(* IEC 61131-3 sources: SRCI/RobotLibrary/Library/POUs/Additional/MC_UnitMeasurement, 1 file *)

(* ---- MC_UnitMeasurementFB.st ---- *)
/// Measure the length of objects in the cartesian space, execution time for specified section of a job or signal output time of a specified signal
FUNCTION_BLOCK MC_UnitMeasurementFB EXTENDS RobotLibraryBaseEnableFB
// -------------------------------------------------------------------------
//  SRCI Robot Library
// -------------------------------------------------------------------------
//
//  Object:      UnitMeasurementFB
//  Author:      Thorsten Brach
//  Date:        2024-06-01
//
//  Description:
//
//
//  Copyright:
//    (C) 2024 Thorsten Brach. All rights reserved
//             Licensed under the LGPL-3.0 license.
//
//  Disclaimer:
//    This project is provided without any guarantee and can be used for
//    private and commercial purposes. Any use is at the user’s
//    own risk and responsibility.
//
// -------------------------------------------------------------------------
VAR_INPUT
  /// command results
  ParCmd            : UnitMeasurementParCmd;
END_VAR

VAR_OUTPUT
  /// Command is transferred and confirmed by the RC
  CommandBuffered   : BOOL;
  /// Receiving of input parameter values has been acknowledged by RC
  ParameterAccepted : BOOL;
  /// command results
  OutCmd            : UnitMeasurementOutCmd;
END_VAR

VAR
  /// internal copy of command parameter
 _parCmd            : UnitMeasurementParCmd;
  /// command data to send
 _command           : UnitMeasurementSendData;
  /// response data received
 _response          : UnitMeasurementRecvData;
  /// measurement number
 _measurementNo     : USINT;
END_VAR

  SUPER^(AxesGroup := AxesGroup);

END_FUNCTION_BLOCK

METHOD INTERNAL CheckAddParameter : BOOL
VAR_INPUT
  /// Payload pointer
  PayloadPtr : UDINT;
END_VAR
VAR
  /// Payload as byte array
  Payload    : ARRAY [1..SIZEOF(_command)] OF BYTE;
  /// Null Byte array
  Null       : ARRAY [1..SIZEOF(_command)] OF BYTE;
  /// Data length to compare
  DataLen    : UDINT;
END_VAR

  // Payload pointer must be decreased by one byte, because ADR(Payload) is already one byte !
  PayloadPtr := LIMIT (0, PayloadPtr - 1, SIZEOF(Payload) -1);
  // Convert command struct to payload array
  SysDepMemCpy( pDest := ADR(Payload), pSrc := ADR(_command), DataLen := SIZEOF(_command));
  // Calculate the data length to compare - at least one byte must be compared !
  DataLen := LIMIT(1, SIZEOF(Payload) - PayloadPtr, SIZEOF(Payload));
  // Compare Payload-Array with Null-Byte-Array
  CheckAddParameter := SysDepMemCmp( pData1 := ADR(Payload) + PayloadPtr , pData2 := ADR(Null), DataLen := DataLen) <>  RobotLibraryConstants.OK ;

END_METHOD

METHOD PROTECTED CheckFunctionSupported : BOOL
VAR_IN_OUT
  /// Robot assignment of function
  AxesGroup : AxesGroup;
END_VAR

  CheckFunctionSupported := AxesGroup.State.RobotData.RCSupportedFunctions.UnitMeasurement;

  IF ( NOT CheckFunctionSupported )
  THEN
    // call base implementation for set error and create log entry
    SUPER^.CheckFunctionSupported(AxesGroup := AxesGroup);
  END_IF

END_METHOD

METHOD PROTECTED CheckParameterChanged : BOOL
VAR_IN_OUT
  /// Robot assignment of function
  AxesGroup    : AxesGroup;
END_VAR

  // Check ParCmd Size is > 0, because MemCmp does not work correctly with size = 0
  IF (SIZEOF(ParCmd) = 0) OR (_stepCmd = 0)
  THEN
    RETURN;
  END_IF

  // compare memory
  _parameterChanged := ( SysDepMemCmp(pData1 := ADR(ParCmd), pData2 := ADR(_parCmd), DataLen := SIZEOF(ParCmd)) <> RobotLibraryConstants.OK );

  // check parameter valid ?
  _parameterValid   := CheckParameterValid( AxesGroup := AxesGroup );

  IF ((  _parameterChanged        )  AND
      (  _parameterValid          )) OR
      (  _parameterUpdateInternal )
  THEN
    // reset internal flag for send parameter update
   _parameterUpdateInternal := FALSE;
    // update internal copy of parameters
   _parCmd := ParCmd;
    // inc parameter sequence
   _command.ParSeq := _command.ParSeq + 1;
    // update command data
    CommandData := CreateCommandPayload(AxesGroup := AxesGroup); // ( Access via reference to rCommandFB in ACR )
    // notify active command register
    AxesGroup.Acyclic.ActiveCommandRegister.NotifyParameterChanged := _uniqueID;
    // Reset parameter accepted flag
    ParameterAccepted := FALSE;
  END_IF

END_METHOD

METHOD PROTECTED CheckParameterValid : BOOL
VAR_IN_OUT
  /// Robot assignment of function
  AxesGroup : AxesGroup;
END_VAR

  CheckParameterValid := TRUE;

  // Check ParCmd.TriggerMode valid ?
  IF (( ParCmd.TriggerMode <> TriggerModeMeasurement.NO_TRIGGER                   ) AND
      ( ParCmd.TriggerMode <> TriggerModeMeasurement.POSITIVE_START_NEGATIVE_STOP ) AND
      ( ParCmd.TriggerMode <> TriggerModeMeasurement.POSITIVE_START_STOP          ))
  THEN
    // Parameter not valid
    CheckParameterValid := FALSE;
    // Set error
    ErrorID := RobotLibraryErrorIdEnum.ERR_TRIGGERMODE_NOT_ALLOWED;
    // Create log entry
    CreateLogMessagePara1 ( Timestamp   := AxesGroup.State.SystemTime,
                            MessageType := MessageType.CMD,
                            Severity    := Severity.ERROR,
                            MessageCode := ErrorID,
                            MessageText := 'Invalid Parameter ParCmd.TriggerMode = {1}',
                            Para1       := TRIGGER_MODE_MEASUREMENT_TO_STRING(ParCmd.TriggerMode));
    RETURN;
  END_IF

  // Check ParCmd.NewMeasurement valid ?
  // -> no plausibility check for boolean

  // Check ParCmd.MeasuringMode valid ?
  IF (( ParCmd.MeasuringMode <> MeasuringUnitMode.VECTOR_LENGTH  ) AND
      ( ParCmd.MeasuringMode <> MeasuringUnitMode.SEGMENT_LENGTH ) AND
      ( ParCmd.MeasuringMode <> MeasuringUnitMode.TIME_DURATION  ))
  THEN
    // Parameter not valid
    CheckParameterValid := FALSE;
    // Set error
    ErrorID := RobotLibraryErrorIdEnum.ERR_PROCESSINGMODE_NOT_ALLOWED;
    // Create log entry
    CreateLogMessagePara1 ( Timestamp   := AxesGroup.State.SystemTime,
                            MessageType := MessageType.CMD,
                            Severity    := Severity.ERROR,
                            MessageCode := ErrorID,
                            MessageText := 'Invalid Parameter ParCmd.MeasuringMode = {1}',
                            Para1       := MEASURING_UNIT_MODE_TO_STRING(ParCmd.MeasuringMode));
    RETURN;
  END_IF

  // Check ParCmd.ListenerID valid ?
  IF (( ParCmd.ListenerID <   0 ) OR
      ( ParCmd.ListenerID > 127 ))
  THEN
    // Parameter not valid
    CheckParameterValid := FALSE;
    // Set error
    ErrorID := RobotLibraryErrorIdEnum.ERR_LISTENERID_MUST_BE_POSITIVE;
    // Create log entry
    CreateLogMessagePara1 ( Timestamp   := AxesGroup.State.SystemTime,
                            MessageType := MessageType.CMD,
                            Severity    := Severity.ERROR,
                            MessageCode := ErrorID,
                            MessageText := 'Invalid Parameter ParCmd.ListenerID = {1}',
                            Para1       := SINT_TO_STRING(ParCmd.ListenerID));
    RETURN;
  END_IF

END_METHOD

METHOD INTERNAL CreateCommandPayload : RobotLibraryCommandDataFB
VAR_IN_OUT
  /// Robot assignment of function
  AxesGroup : AxesGroup;
END_VAR
VAR
  /// internal index for loops
 _idx          : DINT;
  /// Parameter count
 _parameterCnt : DINT;
END_VAR
// Table 6-803: Sent CMD payload (PLC to RC) of "UnitMeasurement"
// --------------------------
// Header
// --------------------------
// Byte 00 : UINT  - Type HB
// Byte 01 :       - Type LB
// Byte 02 : USINT - Reserve | ExecutionMode
// Byte 03 : USINT - ParSeq  | Priority
// --------------------------
// Datablock
// --------------------------
// Byte 04 : SINT   - EmitterID[0]
// Byte 05 : SINT   - EmitterID[1]
// Byte 06 : SINT   - EmitterID[2]
// Byte 07 : SINT   - EmitterID[3]
// Byte 08 : SINT   - ListenerID
// Byte 09 : BYTE   - Reserved
// Byte 10 : USINT  - TriggerMode
// Byte 11 : USINT  - MeasurementNo
// Byte 12 : USINT  - MeasuringMode

  // set command parameter
  _command.CmdTyp          :=  CmdType.UnitMeasurement;
  _command.ExecMode        :=  ExecMode;
  _command.ParSeq          := _command.ParSeq;
  _command.Priority        :=  Priority;
  _command.EmitterID[0]    :=  0;
  _command.EmitterID[1]    :=  0;
  _command.EmitterID[2]    :=  0;
  _command.EmitterID[3]    :=  0;
  _command.ListenerID      :=  _parCmd.ListenerID;
  _command.Reserve         :=  0;
  _command.TriggerMode     :=  _parCmd.TriggerMode;
  _command.MeasurementNo   :=  _measurementNo;
  _command.MeasuringMode   :=  _parCmd.MeasuringMode;

  // copy command data to header
  _cmdHeader := _command;
  // call base implementation to copy header to payload buffer
  CreateCommandPayload := SUPER^.CreateCommandPayload(AxesGroup := AxesGroup);

  FOR _idx := 0 TO 3
  DO
    // Check parameter must be added ?
    IF ( CheckAddParameter(CreateCommandPayload.PayloadPtr))
    THEN
      // add command.EmitterID[x]
      CreateCommandPayload.AddSint(_command.EmitterID[_idx]);
      // inc parameter counter
     _parameterCnt := _parameterCnt + 1;
    END_IF
  END_FOR

  // Check parameter must be added ?
  IF ( CheckAddParameter(CreateCommandPayload.PayloadPtr))
  THEN
    // add command.ListenerID
    CreateCommandPayload.AddSint(_command.ListenerID);
    // inc parameter counter
   _parameterCnt := _parameterCnt + 1;
  END_IF

  // Check parameter must be added ?
  IF ( CheckAddParameter(CreateCommandPayload.PayloadPtr))
  THEN
    // add command.Reserved
    CreateCommandPayload.AddByte(_command.Reserve);
    // inc parameter counter
   _parameterCnt := _parameterCnt + 1;
  END_IF

  // Check parameter must be added ?
  IF ( CheckAddParameter(CreateCommandPayload.PayloadPtr))
  THEN
    // add command.TriggerMode
    CreateCommandPayload.AddUsint(_command.TriggerMode);
    // inc parameter counter
   _parameterCnt := _parameterCnt + 1;
  END_IF

  // Check parameter must be added ?
  IF ( CheckAddParameter(CreateCommandPayload.PayloadPtr))
  THEN
    // add command.MeasurementNo
    CreateCommandPayload.AddUsint(_command.MeasurementNo);
    // inc parameter counter
   _parameterCnt := _parameterCnt + 1;
  END_IF

  // Check parameter must be added ?
  IF ( CheckAddParameter(CreateCommandPayload.PayloadPtr))
  THEN
    // add command.MeasuringMode
    CreateCommandPayload.AddUsint(_command.MeasuringMode);
    // inc parameter counter
   _parameterCnt := _parameterCnt + 1;
  END_IF

  // Create logging
  CreateCommandPayloadLog(AxesGroup := AxesGroup, ParameterCnt := _parameterCnt);

END_METHOD

METHOD INTERNAL CreateCommandPayloadLog
VAR_IN_OUT
  /// Robot assignment of function
  AxesGroup : AxesGroup;
END_VAR
VAR_INPUT
  /// Parameter count
  ParameterCnt : DINT;
END_VAR
VAR
  /// internal index for loops
 _idx : DINT;
END_VAR

  // Create log entry for Parameter start
  CreateLogMessagePara1 ( Timestamp   := AxesGroup.State.SystemTime,
                          MessageType := MessageType.CMD,
                          Severity    := Severity.DEBUG,
                          MessageCode := 0,
                          MessageText := 'Create command payload with the {1} parameter(s) :',
                          Para1       := DINT_TO_STRING(ParameterCnt));

  // Create log entry for EmitterID[x]
  FOR _idx := 0 TO 3
  DO
  // Return if no parameter is remaining...
    IF ( ParameterCnt = 0 ) THEN RETURN; END_IF
    // dec remaining parameter(s)
    ParameterCnt := ParameterCnt - 1;
    // Create log entry for command.EmitterID
    CreateLogMessagePara2 ( Timestamp   := AxesGroup.State.SystemTime,
                            MessageType := MessageType.CMD,
                            Severity    := Severity.DEBUG,
                            MessageCode := 0,
                            MessageText := 'Command.EmitterID[{2}] = {1}',
                            Para1       :=  SINT_TO_STRING(_command.EmitterID[_idx]),
                            Para2       :=  DINT_TO_STRING(_idx));
  END_FOR

  // Return if no parameter is remaining...
  IF ( ParameterCnt = 0 ) THEN RETURN; END_IF
  // dec remaining parameter(s)
  ParameterCnt := ParameterCnt - 1;
  // Create log entry for ListenerID
  CreateLogMessagePara1 ( Timestamp   := AxesGroup.State.SystemTime,
                          MessageType := MessageType.CMD,
                          Severity    := Severity.DEBUG,
                          MessageCode := 0,
                          MessageText := 'Command.ListenerID = {1}',
                          Para1       :=  SINT_TO_STRING(_command.ListenerID));

  // Return if no parameter is remaining...
  IF ( ParameterCnt = 0 ) THEN RETURN; END_IF
  // dec remaining parameter(s)
  ParameterCnt := ParameterCnt - 1;
  // Create log entry for Reserve
  CreateLogMessagePara1 ( Timestamp   := AxesGroup.State.SystemTime,
                          MessageType := MessageType.CMD,
                          Severity    := Severity.DEBUG,
                          MessageCode := 0,
                          MessageText := 'Command.Reserve = {1}',
                          Para1       :=  BYTE_TO_STRING(_command.Reserve));

  // Return if no parameter is remaining...
  IF ( ParameterCnt = 0 ) THEN RETURN; END_IF
  // dec remaining parameter(s)
  ParameterCnt := ParameterCnt - 1;
  // Create log entry for TriggerMode
  CreateLogMessagePara1 ( Timestamp   := AxesGroup.State.SystemTime,
                          MessageType := MessageType.CMD,
                          Severity    := Severity.DEBUG,
                          MessageCode := 0,
                          MessageText := 'Command.TriggerMode = {1}',
                          Para1       :=  TRIGGER_MODE_MEASUREMENT_TO_STRING(_command.TriggerMode));

  // Return if no parameter is remaining...
  IF ( ParameterCnt = 0 ) THEN RETURN; END_IF
  // dec remaining parameter(s)
  ParameterCnt := ParameterCnt - 1;
  // Create log entry for MeasurementNo
  CreateLogMessagePara1 ( Timestamp   := AxesGroup.State.SystemTime,
                          MessageType := MessageType.CMD,
                          Severity    := Severity.DEBUG,
                          MessageCode := 0,
                          MessageText := 'Command.MeasurementNo = {1}',
                          Para1       :=  USINT_TO_STRING(_command.MeasurementNo));

  // Return if no parameter is remaining...
  IF ( ParameterCnt = 0 ) THEN RETURN; END_IF
  // dec remaining parameter(s)
  ParameterCnt := ParameterCnt - 1;
  // Create log entry for MeasuringMode
  CreateLogMessagePara1 ( Timestamp   := AxesGroup.State.SystemTime,
                          MessageType := MessageType.CMD,
                          Severity    := Severity.DEBUG,
                          MessageCode := 0,
                          MessageText := 'Command.MeasuringMode = {1}',
                          Para1       :=  MEASUREING_UNIT_MODE_TO_STRING(_command.MeasuringMode));

END_METHOD

METHOD FB_init : BOOL
VAR_INPUT
  /// if TRUE, the retain variables are initialized (warm start / cold start)
  bInitRetains : BOOL;
  /// if TRUE, the instance afterwards gets moved into the copy code (online change)
  bInCopyCode  : BOOL;
END_VAR

  MyType := 'MC_UnitMeasurementFB';

  ExecMode := ExecutionMode.PARALLEL;
  Priority := PriorityLevel.NORMAL;

END_METHOD

METHOD Protected OnExecCancel : DINT
VAR_IN_OUT
  /// Robot assignment of function
  AxesGroup : AxesGroup;
END_VAR
VAR
  /// internal return value
 _retVal    : DINT;
END_VAR

  OnExecCancel := RobotLibraryConstants.RUNNING;

  CASE _stepCancel OF

    0: // set busy flag
       Busy := TRUE;

       // Create log entry
       CreateLogMessagePara1 ( Timestamp   := AxesGroup.State.SystemTime,
                               MessageType := MessageType.CMD,
                               Severity    := Severity.DEBUG,
                               MessageCode := 0,
                               MessageText := 'Execution of {1} cancled ',
                               Para1       := MyType);

       // try to remove cmd
      _retVal := AxesGroup.Acyclic.ActiveCommandRegister.RemoveCmd(_uniqueID);

       // check result of removement
       IF ( _retVal = RobotLibraryConstants.OK )
       THEN
         // Reset step counter
        _stepCancel := 0;
         // finished okay
         OnExecCancel := RobotLibraryConstants.OK;

         // Create log entry
         CreateLogMessagePara1 ( Timestamp   := AxesGroup.State.SystemTime,
                                 MessageType := MessageType.CMD,
                                 Severity    := Severity.DEBUG,
                                 MessageCode := 0,
                                 MessageText := '{1} successfully removed from ACR',
                                 Para1       := MyType);
       ELSE
         // set timeout
         SetTimeout(PT := _timeoutCancel, rTimer := _timerCancel);
         // inc step counter
        _stepCancel := _stepCancel + 1;

         // Create log entry
         CreateLogMessagePara1 ( Timestamp   := AxesGroup.State.SystemTime,
                                 MessageType := MessageType.CMD,
                                 Severity    := Severity.DEBUG,
                                 MessageCode := 0,
                                 MessageText := '{1} was not removed from ACR because execution was already in progress',
                                 Para1       := MyType);
       END_IF

   1:  // call clear error
       OnExecCancel := OnExecErrorClear(AxesGroup := AxesGroup);

       IF ( OnExecCancel = RobotLibraryConstants.OK)
       THEN
         // Reset busy flag
         Busy := FALSE;
         // Reset step counter
        _stepCancel := 0;
         // finished okay
         OnExecCancel := RobotLibraryConstants.OK;
       END_IF

  ELSE
    // invalid step
    ErrorID := RobotLibraryErrorIdEnum.ERR_INVALID_STEP;
  END_CASE

  // reset step counter
  IF (OnExecCancel <> RobotLibraryConstants.RUNNING)
  THEN
    // Reset FB variables
    Reset();
    // Reset step counter
   _stepCancel := 0;
  END_IF

END_METHOD

METHOD PROTECTED OnExecErrorClear : DINT
VAR_IN_OUT
  /// Robot assignment of function
  AxesGroup : AxesGroup;
END_VAR

  OnExecErrorClear := RobotLibraryConstants.RUNNING;

  CASE _stepClearError OF

    0:  // set busy flag
        Busy := TRUE;
        // trigger parameter update to disable FB
       _parameterUpdateInternal := TRUE;
        // call Check Parameter changed method to trigger the parameter update to disable the function
        CheckParameterChanged(AxesGroup := AxesGroup);
        // set timeout
        SetTimeout(PT := _timeoutClearError, rTimer := _timerClearError);
        // inc step counter
       _stepClearError := _stepClearError + 1;

    1: IF ( _responseReceived )
       THEN
         // reset response received flag
        _responseReceived := FALSE;
         // reset step counter
        _stepClearError := 0;
         // finished
         OnExecErrorClear := RobotLibraryConstants.OK;
       ELSE
         // timeout exceeded ?
         IF (CheckTimeout(_timerClearError) = RobotLibraryConstants.OK)
         THEN
           OnExecErrorClear := RobotLibraryConstants.HAS_ERROR;
         END_IF
  	   END_IF
  ELSE
    // invalid step
    ErrorID := RobotLibraryErrorIdEnum.ERR_INVALID_STEP;
  END_CASE

  // reset step counter
  IF (OnExecErrorClear <> RobotLibraryConstants.RUNNING)
  THEN
    // Reset
    Reset();
    // reset step counter
   _stepClearError := 0;
  END_IF

END_METHOD

METHOD PROTECTED OnExecRun : DINT
VAR_IN_OUT
  /// Robot assignment of function
  AxesGroup : AxesGroup;
END_VAR

  // call base implementation
  SUPER^.OnExecRun(AxesGroup := AxesGroup);

  CASE _stepCmd OF

    00:  IF ( _enable_R.Q ) AND ( NOT Error)
         THEN
           // reset the rising edge
          _enable_R();

           // Check function is supported and parameter are valid ?
           IF (( CheckFunctionSupported( AxesGroup := AxesGroup )) AND
               ( CheckParameterValid   ( AxesGroup := AxesGroup )))
           THEN
             // Reset all internal flags
             Reset();
             // set busy flag
             Busy := TRUE;
             // Reset command outputs
             SysDepMemSet(pDest := ADR(OutCmd), Value := 0, DataLen := SIZEOF(OutCmd));
             // inc measurement number
            _measurementNo := _measurementNo + 1;
             // apply command parameter
            _parCmd := ParCmd;
             // init parameter sequence
            _command.ParSeq := 1;
             // create command data
             CommandData := CreateCommandPayload(AxesGroup := AxesGroup);
             // Add command to active command register
            _uniqueID := AxesGroup.Acyclic.ActiveCommandRegister.AddCmd( pCommandFB := ADR(THIS^ ));
             // set timeout
             SetTimeout(PT := _timeoutCmd, rTimer := _timerCmd);
             // inc step counter
            _stepCmd := _stepCmd + 1;
           END_IF
         END_IF

    01:  // Wait for responce received
         IF ( _responseReceived )
         THEN
           // reset response received flag
          _responseReceived := FALSE;

           CASE  _response.State
           OF
             CmdMessageState.BUFFERED    : CommandBuffered    := TRUE;
             CmdMessageState.ACTIVE      : ParameterAccepted  := TRUE;
                                           Enabled            := TRUE;  {warning 'ToDo: Indicator for Enabled'}
             CmdMessageState.ERROR       : Error              := TRUE;
           END_CASE

           // Update results
           OutCmd.MeasurementActive := _response.MeasurementActive;
           OutCmd.Result            := _response.Result;
           OutCmd.OriginID          := _response.OriginID;
           OutCmd.InvocationCounter := _response.InvocationCounter;

           // Enabled or Error ? -> Reset Busy flag
           IF (( Enabled ) OR
               ( Error   ))
           THEN
             Busy := FALSE;
  				 END_IF

         END_IF

         // do not abort directly, so that the ParSeq update can be send
         IF ( _enable_F.Q )
         THEN
           // Set Busy flag
           Busy := TRUE;
           // trigger parameter update to disable FB
          _parameterUpdateInternal := TRUE;
           // reset the falling edge
          _enable_F();
           // set timeout
           SetTimeout(PT := _timeoutCmd, rTimer := _timerCmd);
           // inc step counter
          _stepCmd := _stepCmd + 1;
         END_IF

        // Wait for response received or timeout or not Initialized
    02: IF ((    _responseReceived                                   )  OR
            (     CheckTimeout(_timerCmd) = RobotLibraryConstants.OK )) OR
           (( NOT AxesGroup.State.Initialized                        )  AND
            ( NOT AxesGroup.State.Synchronized                       ))
        THEN
          Reset();
  	    END_IF

  ELSE
    // invalid step
    ErrorID := RobotLibraryErrorIdEnum.ERR_INVALID_STEP;
  END_CASE

  // Reset FB
  IF (( _enable_R.Q ) OR
      ( _enable_F.Q ))
  THEN
    Reset();
  END_IF

END_METHOD

METHOD INTERNAL ParseResponsePayload : DINT
VAR_INPUT
  /// Response data
  ResponseData : RobotLibraryResponseDataFB;
  /// Timestamp
  Timestamp    : SystemTime;
END_VAR
VAR
  /// Parameter count
 _parameterCnt : DINT;
END_VAR
// Table 6-804: Received CMD payload (RC to PLC) of "UnitMeasurement"
// --------------------------
// Header
// --------------------------
// Byte 00 : USINT - ParSeq | State
// Byte 01 : SINT  - AlarmMessageSeverity
// Byte 02 : UINT  - AlarmMessageCode HB
// Byte 03 :       - AlarmMessageCode LB
// --------------------------
// Datablock
// --------------------------
// Byte 04 : USINT  - InvocationCounter
// Byte 05 : SINT   - Reserved
// Byte 06 : INT    - OriginID HW HB
// Byte 07 :        - OriginID HW LB
// Byte 08 : REAL   - Result HW HB
// Byte 09 :        - Result HW LB
// Byte 10 :        - Result LW HB
// Byte 11 :        - Result LW LB
// Byte 12 : BOOL   - MeasurementActive
// Byte 13 : USINT  - ResultNo
// --------------------------

  // call base implementation to parse the header from payload buffer
  ResponseData.PayloadPtr := SUPER^.ParseResponsePayload(ResponseData := ResponseData, Timestamp := Timestamp);

  // copy parsed header to response
  _response.ParSeq               := _rspHeader.ParSeq;
  _response.State                := _rspHeader.State;
  _response.AlarmMessageSeverity := _rspHeader.AlarmMessageSeverity;
  _response.AlarmMessageCode     := _rspHeader.AlarmMessageCode;

  // Check payload remaining ?
  IF ( ResponseData.IsPayloadRemaining)
  THEN
    // Get Response.InvocationCounter
   _response.InvocationCounter := ResponseData.GetUsint();
    // inc parameter counter
   _parameterCnt := _parameterCnt + 1;
  END_IF

  // Check payload remaining ?
  IF ( ResponseData.IsPayloadRemaining)
  THEN
    // Get Response.Reserve
   _response.Reserve := ResponseData.GetSint();
    // inc parameter counter
   _parameterCnt := _parameterCnt + 1;
  END_IF

  // Check payload remaining ?
  IF ( ResponseData.IsPayloadRemaining)
  THEN
    // Get Response.OriginID
   _response.OriginID := ResponseData.GetInt();
    // inc parameter counter
   _parameterCnt := _parameterCnt + 1;
  END_IF

  // Check payload remaining ?
  IF ( ResponseData.IsPayloadRemaining)
  THEN
    // Get Response.Result
   _response.Result := ResponseData.GetReal();
    // inc parameter counter
   _parameterCnt := _parameterCnt + 1;
  END_IF

  // Check payload remaining ?
  IF ( ResponseData.IsPayloadRemaining)
  THEN
    // Get Response.MeasurementActive
   _response.MeasurementActive := ResponseData.GetBool();
    // inc parameter counter
   _parameterCnt := _parameterCnt + 1;
  END_IF

  // Check payload remaining ?
  IF ( ResponseData.IsPayloadRemaining)
  THEN
    // Get Response.ResultNo
   _response.ResultNo := ResponseData.GetUsint();
    // inc parameter counter
   _parameterCnt := _parameterCnt + 1;
  END_IF

  // Create logging
  ParseResponsePayloadLog(ResponseData := ResponseData, Timestamp := Timestamp, ParameterCnt := _parameterCnt);

END_METHOD

METHOD INTERNAL ParseResponsePayloadLog
VAR_INPUT
  /// Response data
  ResponseData : RobotLibraryResponseDataFB;
  /// Timestamp
  Timestamp    : SystemTime;
  /// Parameter count
  ParameterCnt : DINT;
END_VAR

  // Create log entry for Parameter start
  CreateLogMessagePara1 ( Timestamp   := Timestamp,
                          MessageType := MessageType.CMD,
                          Severity    := Severity.DEBUG,
                          MessageCode := 0,
                          MessageText := '{1} parameter(s) to parse from the response data:',
                          Para1       := DINT_TO_STRING(ParameterCnt));

  // Return if no parameter is remaining...
  IF ( ParameterCnt = 0 ) THEN RETURN; END_IF
  // dec remaining parameter(s)
  ParameterCnt := ParameterCnt - 1;
  // Create log entry for InvocationCounter
  CreateLogMessagePara1 ( Timestamp   := Timestamp,
                          MessageType := MessageType.CMD,
                          Severity    := Severity.DEBUG,
                          MessageCode := 0,
                          MessageText := 'Response.InvocationCounter = {1}',
                          Para1       :=  USINT_TO_STRING(_response.InvocationCounter));

  // Return if no parameter is remaining...
  IF ( ParameterCnt = 0 ) THEN RETURN; END_IF
  // dec remaining parameter(s)
  ParameterCnt := ParameterCnt - 1;
  // Create log entry for Reserve
  CreateLogMessagePara1 ( Timestamp   := Timestamp,
                          MessageType := MessageType.CMD,
                          Severity    := Severity.DEBUG,
                          MessageCode := 0,
                          MessageText := 'Response.Reserve = {1}',
                          Para1       :=  SINT_TO_STRING(_response.Reserve));

  // Return if no parameter is remaining...
  IF ( ParameterCnt = 0 ) THEN RETURN; END_IF
  // dec remaining parameter(s)
  ParameterCnt := ParameterCnt - 1;
  // Create log entry for OriginID
  CreateLogMessagePara1 ( Timestamp   := Timestamp,
                          MessageType := MessageType.CMD,
                          Severity    := Severity.DEBUG,
                          MessageCode := 0,
                          MessageText := 'Response.OriginID = {1}',
                          Para1       :=  INT_TO_STRING(_response.OriginID));

  // Return if no parameter is remaining...
  IF ( ParameterCnt = 0 ) THEN RETURN; END_IF
  // dec remaining parameter(s)
  ParameterCnt := ParameterCnt - 1;
  // Create log entry for Result
  CreateLogMessagePara1 ( Timestamp   := Timestamp,
                          MessageType := MessageType.CMD,
                          Severity    := Severity.DEBUG,
                          MessageCode := 0,
                          MessageText := 'Response.Result = {1}',
                          Para1       :=  REAL_TO_STRING(_response.Result));

  // Return if no parameter is remaining...
  IF ( ParameterCnt = 0 ) THEN RETURN; END_IF
  // dec remaining parameter(s)
  ParameterCnt := ParameterCnt - 1;
  // Create log entry for MeasurementActive
  CreateLogMessagePara1 ( Timestamp   := Timestamp,
                          MessageType := MessageType.CMD,
                          Severity    := Severity.DEBUG,
                          MessageCode := 0,
                          MessageText := 'Response.MeasurementActive = {1}',
                          Para1       :=  BOOL_TO_STRING(_response.MeasurementActive));

  // Return if no parameter is remaining...
  IF ( ParameterCnt = 0 ) THEN RETURN; END_IF
  // dec remaining parameter(s)
  ParameterCnt := ParameterCnt - 1;
  // Create log entry for ResultNo
  CreateLogMessagePara1 ( Timestamp   := Timestamp,
                          MessageType := MessageType.CMD,
                          Severity    := Severity.DEBUG,
                          MessageCode := 0,
                          MessageText := 'Response.ResultNo = {1}',
                          Para1       :=  USINT_TO_STRING(_response.ResultNo));

END_METHOD

METHOD PROTECTED Reset : DINT
VAR_INPUT
END_VAR

  Reset := SUPER^.Reset();

  Busy               := FALSE;
  CommandBuffered    := FALSE;
  ParameterAccepted  := FALSE;

END_METHOD
